{attribute 'qualified_only'}
{attribute 'strict'}
TYPE eRestoreMode : 
(
    None := 0,
    (*~
    <docu>
        <summary>
                Activates automatic restore mechanism for all immediate children (direct members).
        </summary>
    </docu>
    ~*)
    AutoRestoreMembers := 10
);
END_TYPE

(* stored: Version 1.1.0.1
   DUT eRestoreMode: Id {8301561c-4174-07b5-10c0-66adbcb58c64} *)
